SUBAPPLICATION Uebung_011b1 (* Numeric Value Input ADD *)
  (* Standard: 61499-2; Description: Copyright (c) 2023 Meisterschulen am Ostbahnhof This program and the accompanying materials are made available under the terms of the Eclipse Public License 2.0 which is available at https://www.eclipse.org/legal/epl-2.0/ SPDX-License-Identifier: EPL-2.0 *)
  (* Version 1.0, 2023-10-23, Franz Höpfinger, Meisterschulen am Ostbahnhof, initial API and implementation and/or initial documentation *)
  PACKAGE Uebungen;
  IMPORT Uebungen::const::UT::DefaultPool::InputNumber_I1;
  IMPORT Uebungen::const::UT::DefaultPool::InputNumber_I2;
  IMPORT Uebungen::const::UT::DefaultPool::OutputNumber_N1;
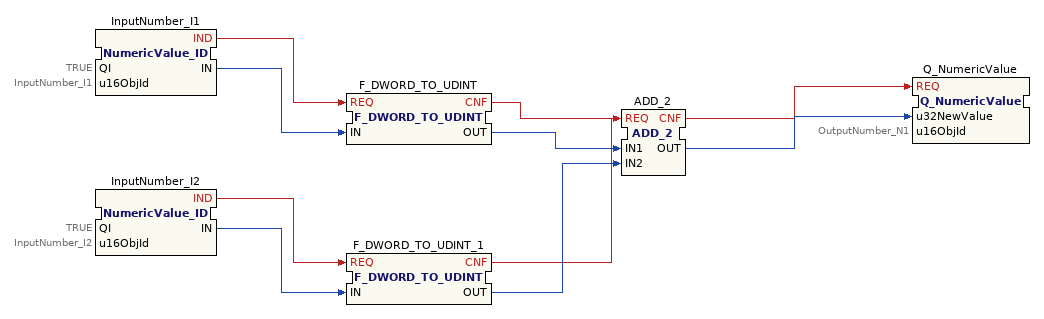
  FBS
    F_DWORD_TO_UDINT : iec61131::conversion::F_DWORD_TO_UDINT;
    InputNumber_I1 : isobus::UT::io::NumericValue::NumericValue_ID(QI := TRUE, u16ObjId := InputNumber_I1);
    Q_NumericValue : isobus::UT::Q::Q_NumericValue(u16ObjId := OutputNumber_N1);
    ADD_2 : iec61131::arithmetic::ADD_2;
    InputNumber_I2 : isobus::UT::io::NumericValue::NumericValue_ID(QI := TRUE, u16ObjId := InputNumber_I2);
    F_DWORD_TO_UDINT_1 : iec61131::conversion::F_DWORD_TO_UDINT;
  END_FBS
  EVENT_CONNECTIONS
    InputNumber_I1.IND TO F_DWORD_TO_UDINT.REQ;
    InputNumber_I2.IND TO F_DWORD_TO_UDINT_1.REQ;
    F_DWORD_TO_UDINT.CNF TO ADD_2.REQ;
    F_DWORD_TO_UDINT_1.CNF TO ADD_2.REQ;
    ADD_2.CNF TO Q_NumericValue.REQ;
  END_CONNECTIONS
  DATA_CONNECTIONS
    InputNumber_I1.IN TO F_DWORD_TO_UDINT.IN;
    InputNumber_I2.IN TO F_DWORD_TO_UDINT_1.IN;
    F_DWORD_TO_UDINT.OUT TO ADD_2.IN1;
    F_DWORD_TO_UDINT_1.OUT TO ADD_2.IN2;
    ADD_2.OUT TO Q_NumericValue.u32NewValue;
  END_CONNECTIONS
END_SUBAPPLICATION
